// SIMATIC S7-200 project (STEP 7-Micro/WIN), CPU 222 REL 02.01

SYMBOL_TABLE USUARIO1
PULSADOR_PARO    I0.0
PULSADOR_MARCHA  I0.1
LAMPARA          Q0.0
END_SYMBOL_TABLE

ORGANIZATION_BLOCK PRINCIPAL:OB1
TITLE=COMENTARIOS DEL PROGRAMA
BEGIN
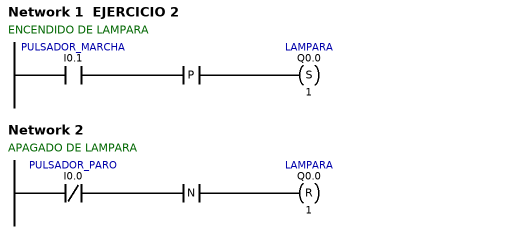
Network 1 // EJERCICIO 2 
// ENCENDIDO DE LAMPARA
// (network saved uncompiled; LAD cells follow)
// row 0: c0 -| |- PULSADOR_MARCHA:I0.1  c1 -|P|-  c2 -(S) LAMPARA:Q0.0, 1
Network 2
// APAGADO DE LAMPARA
// (network saved uncompiled; LAD cells follow)
// row 0: c0 -|/|- PULSADOR_PARO:I0.0  c1 -|N|-  c2 -(R) LAMPARA:Q0.0, 1
END_ORGANIZATION_BLOCK
